TYPE ST_AnalogPressureTemp :
	//Config struct for pressure/temp sensors
STRUCT
	rWarninglevel: REAL;
	rErrorLevel: REAL;
	rPressureMaxSP:REAL;
	rPressureMinSP:REAL;
	rTemperatureMaxSP:REAL;
	rTemperatureMinSP:REAL;
	nRawMax:INT;
	nRawMin:INT;
END_STRUCT
END_TYPE

(* stored: Version 1.1.0.1
   DUT ST_AnalogPressureTemp: Id {442ec741-0c87-4196-8cca-7d8334582bc9} *)
